// Mitsubishi GX Works2 project: De03   PLC: FX2N/FX2NC

PROGRAM MAIN
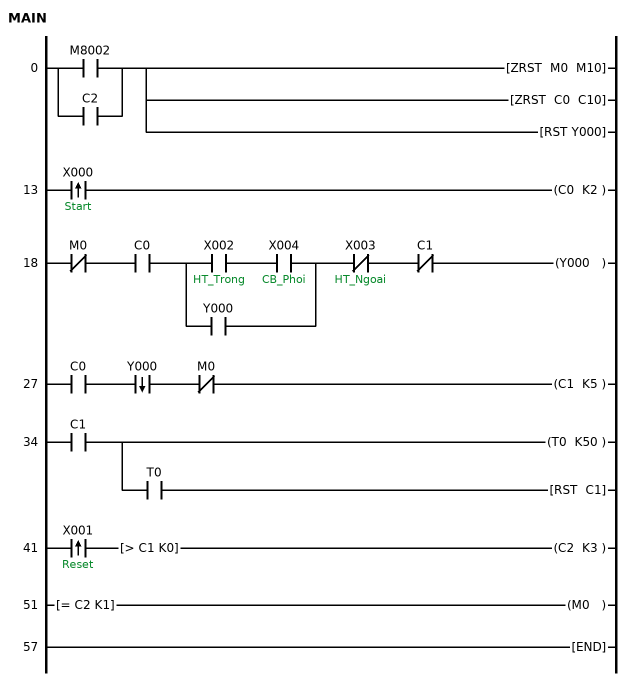
0     LD      M8002
      OR      C2
      ZRST    M0 M10
      ZRST    C0 C10
      RST     Y000
13    LDP     X000  ; Start
      OUT     C0 K2
18    LDI     M0
      AND     C0
      LD      X002  ; HT_Trong
      AND     X004  ; CB_Phoi
      OR      Y000
      ANB
      ANI     X003  ; HT_Ngoai
      ANI     C1
      OUT     Y000
27    LD      C0
      ANDF    Y000
      ANI     M0
      OUT     C1 K5
34    LD      C1
      OUT     T0 K50
      AND     T0
      RST     C1
41    LDP     X001  ; Reset
      AND>    C1 K0
      OUT     C2 K3
51    LD=     C2 K1
      OUT     M0
57    END
END_PROGRAM
